RoboDK station: Basic Trajectory Program.rdk

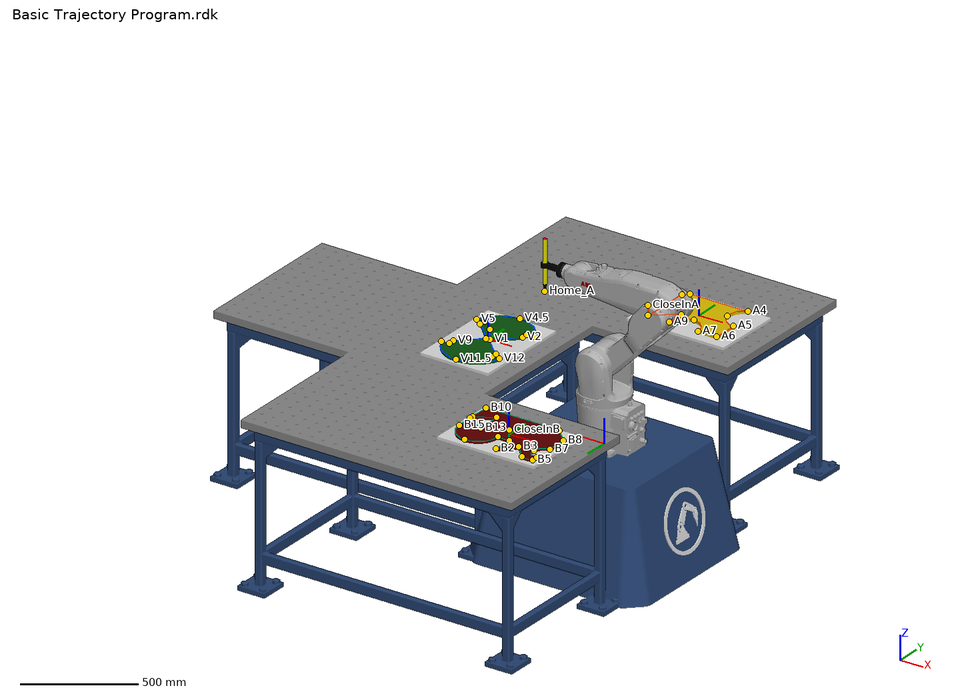
[picture v0: the station drawn from its stored meshes, robots at their saved joint values, targets as dots, program paths as lines]
Station Basic Trajectory Program (saved by RoboDK 5.9.2). Poses are relative to the parent item; angles as X-Y-Z fixed-axis rotations.
  - object Pedestal at (1400, 0, -800) mm, rotated rx 0 ry 0 rz 90 deg, size 844.5 x 933.7 x 500 mm, geometry from Pedestal-H500mm-Type-2.sld
    - frame ABB IRB 1200-5/0.9 Base at (0, 0, 500) mm, rotated rx 0 ry 0 rz 90 deg
      - robot ABB IRB 1200-5/0.9: 6 axes, payload 5 kg, reach 901 mm, repeatability 0.02 mm, weight 52 kg
          modified DH rows (alpha deg, a mm, theta deg, d mm): 0, 0, 0, 399; -90, 0, -90, 0; 0, 448, 0, 0; -90, 42, 0, 451; 90, 0, 0, 0; -90, 0, 180, 82
          joint limits [-170, -100, -200, -270, -130, -360] to [170, 130, 70, 270, 130, 360]; home [0, 0, 0, 0, 0, 0]; saved at [0, -45, 45, 0, 0, 0]
        - tool Tool Lapiz, TCP at (125, 0, 90) mm, size 65 x 250 x 107.5 mm, geometry from Tool Lapiz.IGS
      - target Home_A (Cartesian target) at (306.22, 0, 632.78) mm, rotated rx 0 ry 90 rz 0 deg; joints [0, -45, 45, 0, 0, 0] of ABB IRB 1200-5/0.9
  - folder Trajectories
    - object Trajectory_1 at (1400, 700, 0) mm, rotated rx 90 ry 0 rz 0 deg, size 500 x 25.4 x 350 mm, geometry from trayectoria 1.IGS
    - object Trajectory_3 at (800, 0, 0) mm, rotated rx 0 ry 0 rz 90 deg, size 500 x 350 x 25.4 mm, geometry from trayectoria 3.IGS
    - object Trajectory_2 at (1400, -700, 0) mm, rotated rx 0 ry 0 rz 180 deg, size 500 x 350 x 25.4 mm, geometry from trayectoria 2.IGS
  - folder Tables
    - object Table_1 at (0, 0, 0) mm, size 1420 x 820 x 800 mm, geometry from Table-1400x800x800mm.sld
    - object Table_3 at (700, -800, 0) mm, size 1420 x 820 x 800 mm, geometry from Table-1400x800x800mm.sld
    - object Table_2 at (700, 800, 0) mm, size 1420 x 820 x 800 mm, geometry from Table-1400x800x800mm.sld
  - frame Ref_Trajectory_1 at (800, 0, 25.4) mm
    - target V1 (Cartesian target) at (10, 0, 0) mm, rotated rx 0 ry 90 rz 180 deg; joints [0, 20.261, 39.586, 0, -59.847, 0] of ABB IRB 1200-5/0.9
    - target V2 (Cartesian target) at (110, 100, 0) mm, rotated rx 0 ry 90 rz 180 deg; joints [-17.457, 12.438, 51.354, -19.316, -65.083, 8.4] of ABB IRB 1200-5/0.9
    - target V3 (Cartesian target) at (110, 130, 0) mm, rotated rx 0 ry 90 rz 180 deg; joints [-22.235, 13.414, 49.968, -24.573, -65.497, 10.738] of ABB IRB 1200-5/0.9
    - target V4 (Cartesian target) at (150, 130, 0) mm, rotated rx 0 ry 90 rz 180 deg; joints [-25.062, 9.839, 54.915, -27.339, -67.273, 11.296] of ABB IRB 1200-5/0.9
    - target V4.5 (Cartesian target) at (0, 237.3, 0) mm, rotated rx 0 ry 90 rz 180 deg; joints [-29.006, 26.625, 29.113, -33.856, -60.504, 18.278] of ABB IRB 1200-5/0.9
    - target V5 (Cartesian target) at (-150, 130, 0) mm, rotated rx 0 ry 90 rz -180 deg; joints [-12.676, 35.985, 12.716, -16.666, -49.917, 10.911] of ABB IRB 1200-5/0.9
    - target V6 (Cartesian target) at (-110, 130, 0) mm, rotated rx 0 ry 90 rz -180 deg; joints [-13.584, 32.387, 19.131, -17.154, -52.782, 10.576] of ABB IRB 1200-5/0.9
    - target V7 (Cartesian target) at (-110, 100, 0) mm, rotated rx 0 ry 90 rz -180 deg; joints [-10.53, 31.817, 20.137, -13.28, -52.705, 8.139] of ABB IRB 1200-5/0.9
    - target V8 (Cartesian target) at (-10, 0, 0) mm, rotated rx 0 ry 90 rz -180 deg; joints [0, 22.051, 36.71, 0, -58.761, 0] of ABB IRB 1200-5/0.9
    - target V9 (Cartesian target) at (-110, -100, 0) mm, rotated rx 0 ry 90 rz 180 deg; joints [10.53, 31.817, 20.137, 13.28, -52.705, -8.139] of ABB IRB 1200-5/0.9
    - target V10 (Cartesian target) at (-110, -130, 0) mm, rotated rx 0 ry 90 rz 180 deg; joints [13.584, 32.387, 19.131, 17.154, -52.782, -10.576] of ABB IRB 1200-5/0.9
    - target V11 (Cartesian target) at (-150, -130, 0) mm, rotated rx 0 ry 90 rz -180 deg; joints [12.676, 35.985, 12.716, 16.666, -49.917, -10.911] of ABB IRB 1200-5/0.9
    - target V11.5 (Cartesian target) at (0, -237.3, 0) mm, rotated rx 0 ry 90 rz -180 deg; joints [29.006, 26.625, 29.113, 33.856, -60.504, -18.278] of ABB IRB 1200-5/0.9
    - target V12 (Cartesian target) at (150, -130, 0) mm, rotated rx 0 ry 90 rz -180 deg; joints [25.062, 9.839, 54.915, 27.339, -67.273, -11.296] of ABB IRB 1200-5/0.9
    - target V13 (Cartesian target) at (110, -130, 0) mm, rotated rx 0 ry 90 rz -180 deg; joints [22.235, 13.414, 49.968, 24.573, -65.497, -10.738] of ABB IRB 1200-5/0.9
    - target V14 (Cartesian target) at (110, -100, 0) mm, rotated rx 0 ry 90 rz 180 deg; joints [17.457, 12.438, 51.354, 19.316, -65.083, -8.4] of ABB IRB 1200-5/0.9
    - target CloseInV (Cartesian target) at (10, 0, 50) mm, rotated rx 0 ry 90 rz -180 deg; joints [0, 14.3, 38.291, 0, -52.59, 0] of ABB IRB 1200-5/0.9
  - program Home_position (3 instructions, listed below)
  - program Green_object (19 instructions, listed below)
  - program Main (7 instructions, listed below)
  - frame Ref_Trajectory_2 at (1400, 700, 25) mm
    - target CloseInA (Cartesian target) at (-175, -125, 50) mm, rotated rx 0 ry 90 rz 90 deg; joints [-66.527, 16.532, 35.273, 28.922, -55.447, -17.4] of ABB IRB 1200-5/0.9
    - target A1 (Cartesian target) at (-175, -125, 0) mm, rotated rx 0 ry 90 rz 90 deg; joints [-66.527, 22.22, 36.52, 26.93, -61.577, -13.593] of ABB IRB 1200-5/0.9
    - target A2 (Cartesian target) at (-175, 125, 0) mm, rotated rx 0 ry 90 rz 90 deg; joints [-74.998, 44.217, -2.292, 21.856, -44.055, -16.08] of ABB IRB 1200-5/0.9
    - target A3 (Cartesian target) at (-150, 150, 0) mm, rotated rx 0 ry 90 rz 90 deg; joints [-77.525, 46.147, -5.892, 18.9, -41.827, -14.312] of ABB IRB 1200-5/0.9
    - target A4 (Cartesian target) at (150, 150, 0) mm, rotated rx 0 ry 90 rz 90 deg; joints [-102.475, 46.147, -5.892, -18.9, -41.827, 14.312] of ABB IRB 1200-5/0.9
    - target A4.5 (Cartesian target) at (103.51, 62.7, 0) mm, rotated rx 0 ry 90 rz 90 deg; joints [-99.939, 36.703, 11.491, -13.229, -48.959, 8.775] of ABB IRB 1200-5/0.9
    - target A5 (Cartesian target) at (180, 0, 0) mm, rotated rx 0 ry 90 rz 90 deg; joints [-108.825, 32.822, 18.435, -23.609, -53.676, 14.516] of ABB IRB 1200-5/0.9
    - target A6 (Cartesian target) at (180, -125, 0) mm, rotated rx 0 ry 90 rz 90 deg; joints [-114.068, 22.4, 36.227, -27.616, -61.618, 13.964] of ABB IRB 1200-5/0.9
    - target A7 (Cartesian target) at (85, -125, 0) mm, rotated rx 0 ry 90 rz 90 deg; joints [-101.91, 19.761, 40.467, -13.658, -60.931, 6.733] of ABB IRB 1200-5/0.9
    - target A8 (Cartesian target) at (10, -50, 0) mm, rotated rx 0 ry 90 rz 90 deg; joints [-91.198, 25.665, 30.815, -1.437, -56.488, 0.794] of ABB IRB 1200-5/0.9
    - target A9 (Cartesian target) at (-65, -125, 0) mm, rotated rx 0 ry 90 rz 90 deg; joints [-80.838, 19.432, 40.987, 10.507, -60.833, -5.165] of ABB IRB 1200-5/0.9
    - target A10 (Cartesian target) at (-65, -35, 0) mm, rotated rx 0 ry 90 rz 90 deg; joints [-82.489, 27.37, 27.925, 9.111, -55.634, -5.173] of ABB IRB 1200-5/0.9
  - program Yellow_object (14 instructions, listed below)
  - frame Ref_Trajectory_3 at (1400, -700, 25) mm
    - target CloseInB (Cartesian target) at (35.4, -50.4, 50) mm, rotated rx 0 ry 90 rz -90 deg; joints [93.502, 30.506, 13.803, 5.007, -44.419, -3.581] of ABB IRB 1200-5/0.9
    - target B1 (Cartesian target) at (35.4, -50.4, 0) mm, rotated rx 0 ry 90 rz -90 deg; joints [93.502, 34.813, 14.89, 4.588, -49.794, -2.965] of ABB IRB 1200-5/0.9
    - target B2 (Cartesian target) at (35.4, -149.6, 0) mm, rotated rx 0 ry 90 rz -90 deg; joints [92.991, 44.474, -2.771, 4.49, -41.79, -3.351] of ABB IRB 1200-5/0.9
    - target B3 (Cartesian target) at (102.9, -79.6, 0) mm, rotated rx 0 ry 90 rz -90 deg; joints [99.612, 38.276, 8.64, 13.055, -47.663, -8.876] of ABB IRB 1200-5/0.9
    - target B4 (Cartesian target) at (170.4, -149.6, 0) mm, rotated rx 0 ry 90 rz -90 deg; joints [104.116, 46.609, -6.756, 21.427, -41.883, -16.287] of ABB IRB 1200-5/0.9
    - target B5 (Cartesian target) at (224.6, -149.6, 0) mm, rotated rx 0 ry 90 rz -90 deg; joints [108.338, 48.266, -9.867, 28.086, -41.936, -21.652] of ABB IRB 1200-5/0.9
    - target B6 (Cartesian target) at (224.6, -119.6, 0) mm, rotated rx 0 ry 90 rz -90 deg; joints [109.128, 45.198, -4.119, 27.826, -44.586, -20.601] of ABB IRB 1200-5/0.9
    - target B6.5 (Cartesian target) at (174.9, -69.6, 0) mm, rotated rx 0 ry 90 rz -90 deg; joints [106.313, 38.892, 7.517, 22.003, -48.567, -14.971] of ABB IRB 1200-5/0.9
    - target B7 (Cartesian target) at (224.6, -19.6, 0) mm, rotated rx 0 ry 90 rz -90 deg; joints [112.301, 35.967, 12.818, 28.601, -52.439, -18.386] of ABB IRB 1200-5/0.9
    - target B8 (Cartesian target) at (224.6, 79.6, 0) mm, rotated rx 0 ry 90 rz -90 deg; joints [116.606, 27.748, 27.279, 31.437, -59.17, -17.395] of ABB IRB 1200-5/0.9
    - target B9 (Cartesian target) at (154.6, 149.6, 0) mm, rotated rx 0 ry 90 rz -90 deg; joints [112.223, 19.482, 40.908, 25.17, -62.781, -12.131] of ABB IRB 1200-5/0.9
    - target B10 (Cartesian target) at (-224.6, 149.6, 0) mm, rotated rx 0 ry 90 rz -90 deg; joints [59.309, 22.281, 36.421, -34.785, -63.466, 17.24] of ABB IRB 1200-5/0.9
    - target B11 (Cartesian target) at (-224.6, 49.6, 0) mm, rotated rx 0 ry 90 rz -90 deg; joints [64.851, 30.164, 23.104, -30.361, -57.223, 17.595] of ABB IRB 1200-5/0.9
    - target B12 (Cartesian target) at (-134.6, 99.6, 0) mm, rotated rx 0 ry 90 rz -90 deg; joints [72.558, 23.083, 35.109, -20.29, -59.812, 10.531] of ABB IRB 1200-5/0.9
    - target B13 (Cartesian target) at (-134.6, -20.4, 0) mm, rotated rx 0 ry 90 rz -90 deg; joints [76.21, 33.448, 17.325, -17.58, -52.108, 11.012] of ABB IRB 1200-5/0.9
    - target B14 (Cartesian target) at (-224.6, 29.6, 0) mm, rotated rx 0 ry 90 rz -90 deg; joints [65.742, 31.806, 20.23, -29.752, -55.885, 17.775] of ABB IRB 1200-5/0.9
    - target B15 (Cartesian target) at (-224.6, -50.4, 0) mm, rotated rx 0 ry 90 rz -90 deg; joints [68.778, 38.681, 7.901, -28.129, -50.156, 18.907] of ABB IRB 1200-5/0.9
    - target B15.5 (Cartesian target) at (-124.6, -150.4, 0) mm, rotated rx 0 ry 90 rz -90 deg; joints [79.593, 45.652, -4.968, -15.735, -41.769, 11.867] of ABB IRB 1200-5/0.9
    - target B16 (Cartesian target) at (-24.6, -50.4, 0) mm, rotated rx 0 ry 90 rz -90 deg; joints [87.565, 34.761, 14.983, -3.19, -49.788, 2.061] of ABB IRB 1200-5/0.9
  - program Red_Object (21 instructions, listed below)
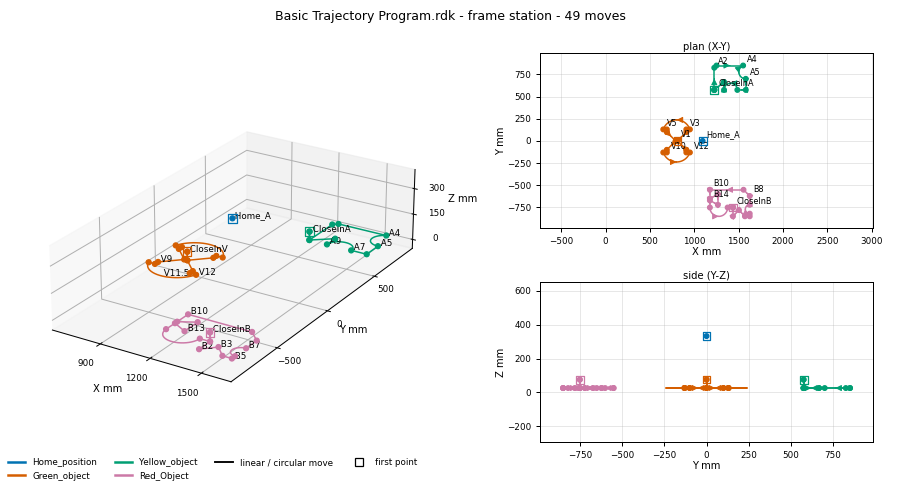
[picture p0: tool path of Basic Trajectory Program.rdk in frame station, 49 of 49 moves have a stored position in this frame; points joined in program order, loops and branches not executed]

--- program Home_position (robot ABB IRB 1200-5/0.9) ---
  Set Ref.: ABB IRB 1200-5/0.9 Base
  Set Tool: Tool Lapiz
  MoveJ (Home_A)

--- program Green_object (robot ABB IRB 1200-5/0.9) ---
  Set Ref.: Ref_Trajectory_1
  Set Tool: Tool Lapiz
  MoveJ (CloseInV)
  MoveL (V1)
  MoveL (V2)
  MoveL (V3)
  MoveL (V4)
  MoveC (V4.5, V5)
  MoveL (V6)
  MoveL (V7)
  MoveL (V8)
  MoveL (V9)
  MoveL (V10)
  MoveL (V11)
  MoveC (V11.5, V12)
  MoveL (V13)
  MoveL (V14)
  MoveL (V1)
  MoveL (CloseInV)

--- program Main (robot ABB IRB 1200-5/0.9) ---
  Call Home_position
  Call Green_object
  Call Home_position
  Call Yellow_object
  Call Home_position
  Call Red_Object
  Call Home_position

--- program Yellow_object (robot ABB IRB 1200-5/0.9) ---
  Set Ref.: Ref_Trajectory_2
  Set Tool: Tool Lapiz
  MoveJ (CloseInA)
  MoveL (A1)
  MoveL (A2)
  MoveL (A3)
  MoveL (A4)
  MoveC (A4.5, A5)
  MoveL (A6)
  MoveL (A7)
  MoveC (A8, A9)
  MoveL (A10)
  MoveL (A1)
  MoveL (CloseInA)

--- program Red_Object (robot ABB IRB 1200-5/0.9) ---
  Set Ref.: Ref_Trajectory_3
  Set Tool: Tool Lapiz
  MoveJ (CloseInB)
  MoveL (B1)
  MoveL (B2)
  MoveL (B3)
  MoveL (B4)
  MoveL (B5)
  MoveL (B6)
  MoveC (B6.5, B7)
  MoveL (B8)
  MoveL (B9)
  MoveL (B10)
  MoveL (B11)
  MoveL (B12)
  MoveL (B13)
  MoveL (B14)
  MoveL (B15)
  MoveC (B15.5, B16)
  MoveL (B1)
  MoveL (CloseInB)
